// TIA Portal project "Saracinesca" (V16)

(* hardware
DEVICE "S7-1200 station_1"  S7-1200 Station
   slot 0: "Telaio di montaggio_0"  S7-1200 Rack  Rack  V1.0
   slot 1: "PLC_1"  CPU 1212C DC/DC/DC  6ES7 212-1AE40-0XB0  V4.1
*)

// ===== PLC "PLC_1"  CPU 1212C DC/DC/DC =====

VAR_GLOBAL   // PLC tag table "Tabella delle variabili standard"
   "S" AT %I0.0 : Bool;
   "FDN" AT %I0.1 : Bool;
   "FUP" AT %I0.2 : Bool;
   "F" AT %I0.3 : Bool;
   "MDN" AT %Q0.1 : Bool;
   "MUP" AT %Q0.2 : Bool;
END_VAR

DATA_BLOCK "VariabiliDiStato"   // DB1
{ S7_Optimized_Access := 'TRUE' }
VERSION : 0.1
   VAR RETAIN
      HOME : Bool := true;
      MOVE_UP : Bool;
      STOP_MOVE_UP : Bool;
      WAIT : Bool;
      MOVE_DOWN : Bool;
   END_VAR
BEGIN
END_DATA_BLOCK

ORGANIZATION_BLOCK "Main"   // OB1, LAD, ProgramCycle
TITLE = "Main Program Sweep (Cycle)"
{ S7_Optimized_Access := 'TRUE' }
VERSION : 0.1
   VAR_INPUT
      Initial_Call : Bool;   // Initial call of this OB
      Remanence : Bool;   // =True, if remanent data are available
   END_VAR
   VAR_TEMP   // added for the SCL form of the ladder/FBD networks
      _w1 : Bool;
   END_VAR
BEGIN

REGION Network 1
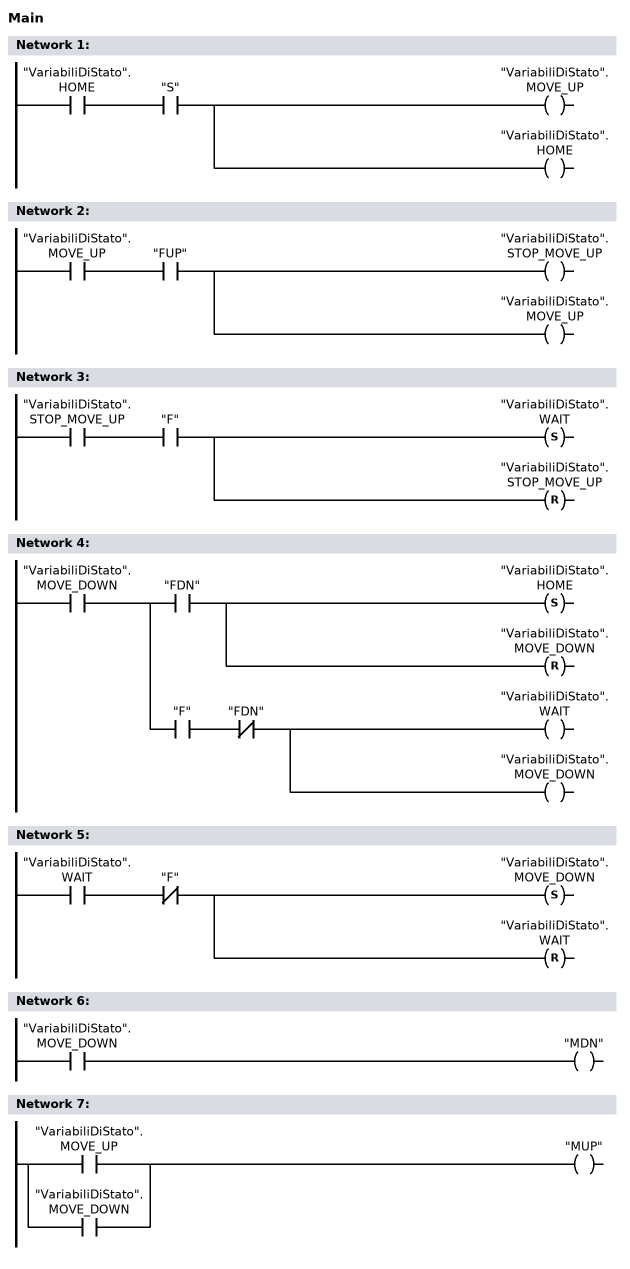
   RUNG wire#powerrail
      Contact( "VariabiliDiStato".HOME )
      Contact( "S" )
      wire#w1
      Coil( "VariabiliDiStato".MOVE_UP )
   END_RUNG
   RUNG wire#w1
      Coil( "VariabiliDiStato".HOME )
   END_RUNG
   // the same network as SCL:
   "VariabiliDiStato".MOVE_UP := "VariabiliDiStato".HOME AND "S";
   "VariabiliDiStato".HOME := "VariabiliDiStato".MOVE_UP;
END_REGION

REGION Network 2
   RUNG wire#powerrail
      Contact( "VariabiliDiStato".MOVE_UP )
      Contact( "FUP" )
      wire#w1
      Coil( "VariabiliDiStato".STOP_MOVE_UP )
   END_RUNG
   RUNG wire#w1
      Coil( "VariabiliDiStato".MOVE_UP )
   END_RUNG
   // the same network as SCL:
   "VariabiliDiStato".STOP_MOVE_UP := "VariabiliDiStato".MOVE_UP AND "FUP";
   "VariabiliDiStato".MOVE_UP := "VariabiliDiStato".STOP_MOVE_UP;
END_REGION

REGION Network 3
   RUNG wire#powerrail
      Contact( "VariabiliDiStato".STOP_MOVE_UP )
      Contact( "F" )
      wire#w1
      S_Coil( "VariabiliDiStato".WAIT )
   END_RUNG
   RUNG wire#w1
      R_Coil( "VariabiliDiStato".STOP_MOVE_UP )
   END_RUNG
   // the same network as SCL:
   IF "VariabiliDiStato".STOP_MOVE_UP AND "F" THEN
       "VariabiliDiStato".WAIT := TRUE;
       "VariabiliDiStato".STOP_MOVE_UP := FALSE;
   END_IF;
END_REGION

REGION Network 4
   RUNG wire#powerrail
      Contact( "VariabiliDiStato".MOVE_DOWN )
      wire#w1
      Contact( "FDN" )
      wire#w2
      S_Coil( "VariabiliDiStato".HOME )
   END_RUNG
   RUNG wire#w2
      R_Coil( "VariabiliDiStato".MOVE_DOWN )
   END_RUNG
   RUNG wire#w1
      Contact( "F" )
      I_Contact( "FDN" )
      wire#w3
      Coil( "VariabiliDiStato".WAIT )
   END_RUNG
   RUNG wire#w3
      Coil( "VariabiliDiStato".MOVE_DOWN )
   END_RUNG
   // the same network as SCL:
   IF "VariabiliDiStato".MOVE_DOWN AND "FDN" THEN "VariabiliDiStato".HOME := TRUE; END_IF;
   #_w1 := "VariabiliDiStato".MOVE_DOWN;
   IF "VariabiliDiStato".MOVE_DOWN AND "FDN" THEN "VariabiliDiStato".MOVE_DOWN := FALSE; END_IF;
   "VariabiliDiStato".WAIT := #_w1 AND "F" AND NOT "FDN";
   "VariabiliDiStato".MOVE_DOWN := "VariabiliDiStato".WAIT;
END_REGION

REGION Network 5
   RUNG wire#powerrail
      Contact( "VariabiliDiStato".WAIT )
      I_Contact( "F" )
      wire#w1
      S_Coil( "VariabiliDiStato".MOVE_DOWN )
   END_RUNG
   RUNG wire#w1
      R_Coil( "VariabiliDiStato".WAIT )
   END_RUNG
   // the same network as SCL:
   IF "VariabiliDiStato".WAIT AND NOT "F" THEN
       "VariabiliDiStato".MOVE_DOWN := TRUE;
       "VariabiliDiStato".WAIT := FALSE;
   END_IF;
END_REGION

REGION Network 6
   RUNG wire#powerrail
      Contact( "VariabiliDiStato".MOVE_DOWN )
      Coil( "MDN" )
   END_RUNG
   // the same network as SCL:
   "MDN" := "VariabiliDiStato".MOVE_DOWN;
END_REGION

REGION Network 7
   RUNG wire#powerrail
      Contact( "VariabiliDiStato".MOVE_UP )
      wire#w1
      Coil( "MUP" )
   END_RUNG
   RUNG wire#powerrail
      Contact( "VariabiliDiStato".MOVE_DOWN )
   END_RUNG wire#w1
   // the same network as SCL:
   "MUP" := "VariabiliDiStato".MOVE_UP OR "VariabiliDiStato".MOVE_DOWN;
END_REGION
END_ORGANIZATION_BLOCK